// TIA Portal V18 export
TYPE "IAI Input Struct"
// stored: IsFailsafeCompliant false
   STRUCT
      "Input 4 word_Man1" : Struct
         "Reserve_0.0" : Bool;   // 网关正常动作时ON
         "Reserve_0.1" : Bool;
         "Reserve_0.2" : Bool;
         "Reserve_0.3" : Bool;
         "Reserve_0.4" : Bool;
         "Reserve_0.5" : Bool;
         "Reserve_0.6" : Bool;
         online : Bool;
         Reserve_Byte_1 : Byte;
         Reserve_Word_2 : Word;
         Reserve_Word_4 : Word;
         Reserve_Word_6 : Word;
      END_STRUCT;
      "Input 4 word_Man2" : Struct
         Reserve_Word_8 : Word;
         Reserve_Word_10 : Word;
         Reserve_Word_12 : Word;
         Reserve_Word_14 : Word;
      END_STRUCT;
      "Input 4 word_1" : Struct
         "Current Position" : DInt;   // 当前位置
         "current value" : DInt;   // 当前马达指令电流值
      END_STRUCT;
      "Input 4 word_2" : Struct
         "Current Speed" : Int;   // 当前速度
         Reserve_12 : Int;
         "Error Code" : Int;   // 报警代码
         MEND : Bool;   // 指令完成
         Reserve_9 : Bool;   // 不能使用
         Reserve_10 : Bool;   // 不能使用
         Reserve_11 : Bool;   // 不能使用
         Zone_1 : Bool;   // 区域输出监视1
         Zone_2 : Bool;   // 区域输出监视2
         CRDY : Bool;   // 控制器准备完成
         EMGS : Bool;   // 紧急停止状态
         Pend : Bool;   // 到位完成
         Hend : Bool;   // 原点复位完成
         Move : Bool;   // 移动中
         ALM : Bool;   // 报警
         SV : Bool;   // 运行准备结束(伺服ON)
         PSFL : Bool;   // 推压动作空转
         Reserve_6 : Bool;   // 不能使用
         ALML : Bool;   // 轻故障报警输出
      END_STRUCT;
   END_STRUCT;
END_TYPE
